{attribute 'qualified_only'}
VAR_GLOBAL
END_VAR

(* stored: Version 1.1.0.1, ProductVersion 3.1.4024.12
   GVL G_FilterConstants: Id {8fda0547-9d0e-42f5-b69f-98e6c021777a} *)
